Staubli VAL3: onExit.pgx

program onExit(bool x_bSave)
  local string l_sEmpty
  local num l_nResult
  local string l_sMessage
begin
  if x_bSave
    // SAVE IT
    l_sEmpty=""
    l_nResult=0
    call prog:save(l_sEmpty,l_nResult)
    call language:message(l_sMessage,-4)
    call use:timerDialog(l_sMessage,1)
  endIf
  sProgType="PROG"
  nProgID=0
end
